{attribute addProperty BoxType "EL3201-0000-0016"}
{attribute addProperty Id "RTD_InputsAT %I*RTD_Inputs_BC62E3BB7290WcStateAT %I*WcState_98A4DF7520.250InfoDataAT %I*InfoData_BC63D37F80100"}
{attribute addProperty CRC "3885355868"}
{attribute addProperty SizeInBites "154"}
{attribute addProperty SizeInBytes "19.25"}
TYPE EL3201_FFA6ACB3 :
STRUCT
	{attribute addProperty Name "RTD_Inputs"}
	RTD_Inputs : RTD_Inputs_BC62E3BB;
	{attribute addProperty Name "WcState"}
	WcState : WcState_98A4DF75;
	{attribute addProperty Name "InfoData"}
	InfoData : InfoData_BC63D37F;
END_STRUCT
END_TYPE

(* stored: Version 1.2.0.0, ProductVersion 3.1.4024.9
   DUT EL3201_FFA6ACB3: Id {a726cd25-a194-4e37-999a-22133ba57c51} *)
